PROGRAM MAIN
VAR
END_VAR

END_PROGRAM

(* stored: Version 1.1.0.1
   POU MAIN: Id {e45175f3-872e-4651-bbfd-cbc74f854a11} *)
